Fanuc KAREL source: kd00027.KL

-- PROVISIONAL review KL for V940-1; original PC SHA256 4958e576c52cb7cb67cc84240dfcc17bb5f9bce8e00d0007067ecd356c9ff9c7
-- Incomplete behavior may be omitted. Consult companion uncertainty JSON. Do not deploy.
PROGRAM KD00027
%NOLOCKGROUP
VAR
  I : INTEGER
  J : INTEGER
  B : BOOLEAN
  R : REAL
  S : STRING[80]
BEGIN
  -- V9_ZERO_TABLE_METADATA_HINT layout=0001; no indexed target words; source/name/runtime held
  -- UNRESOLVED_PC offsets 5-21; opcodes 9D,81,18,9D,12,22,9D,13,04
  -- UNRESOLVED_PC offsets 26-30; opcodes 7F
END KD00027
